FUNCTION_BLOCK ConveyorCTLServer (* Basic Function Block Type *)
  (* Standard: 61499-2 *)
  (* Version 0.2, 2003-12-04, JHC, Rockwell Automation, Renamed for better indexing. *)
  (* Version 0.1, 2002-11-05, JHC, Rockwell Automation, Corrected missing ST element in Algorithm REQ. *)
  (* Version 0.0, 2000-05-30, JHC, Rockwell Automation *)
  (* Compiler header: package fb.rt.cs725; *)
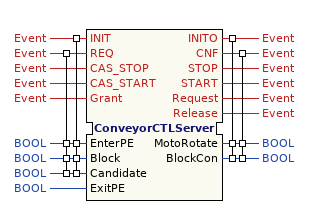
  EVENT_INPUT
    INIT WITH EnterPE, Block, Candidate; (* Initialization Request *)
    REQ WITH EnterPE, Block, Candidate; (* Normal Execution Request *)
    CAS_STOP;
    CAS_START;
    Grant;
  END_EVENT
  EVENT_OUTPUT
    INITO WITH MotoRotate, BlockCon; (* Initialization Confirm *)
    CNF WITH MotoRotate, BlockCon; (* Execution Confirmation *)
    STOP;
    START;
    Request;
    Release;
  END_EVENT
  VAR_INPUT
    EnterPE : BOOL; (* Input event qualifier *)
    Block : BOOL;
    Candidate : BOOL;
    ExitPE : BOOL;
  END_VAR
  VAR_OUTPUT
    MotoRotate : BOOL; (* Output event qualifier *)
    BlockCon : BOOL;
  END_VAR
  VAR
    lastPE : BOOL := 1;
    lastBlock : BOOL := 0;
  END_VAR
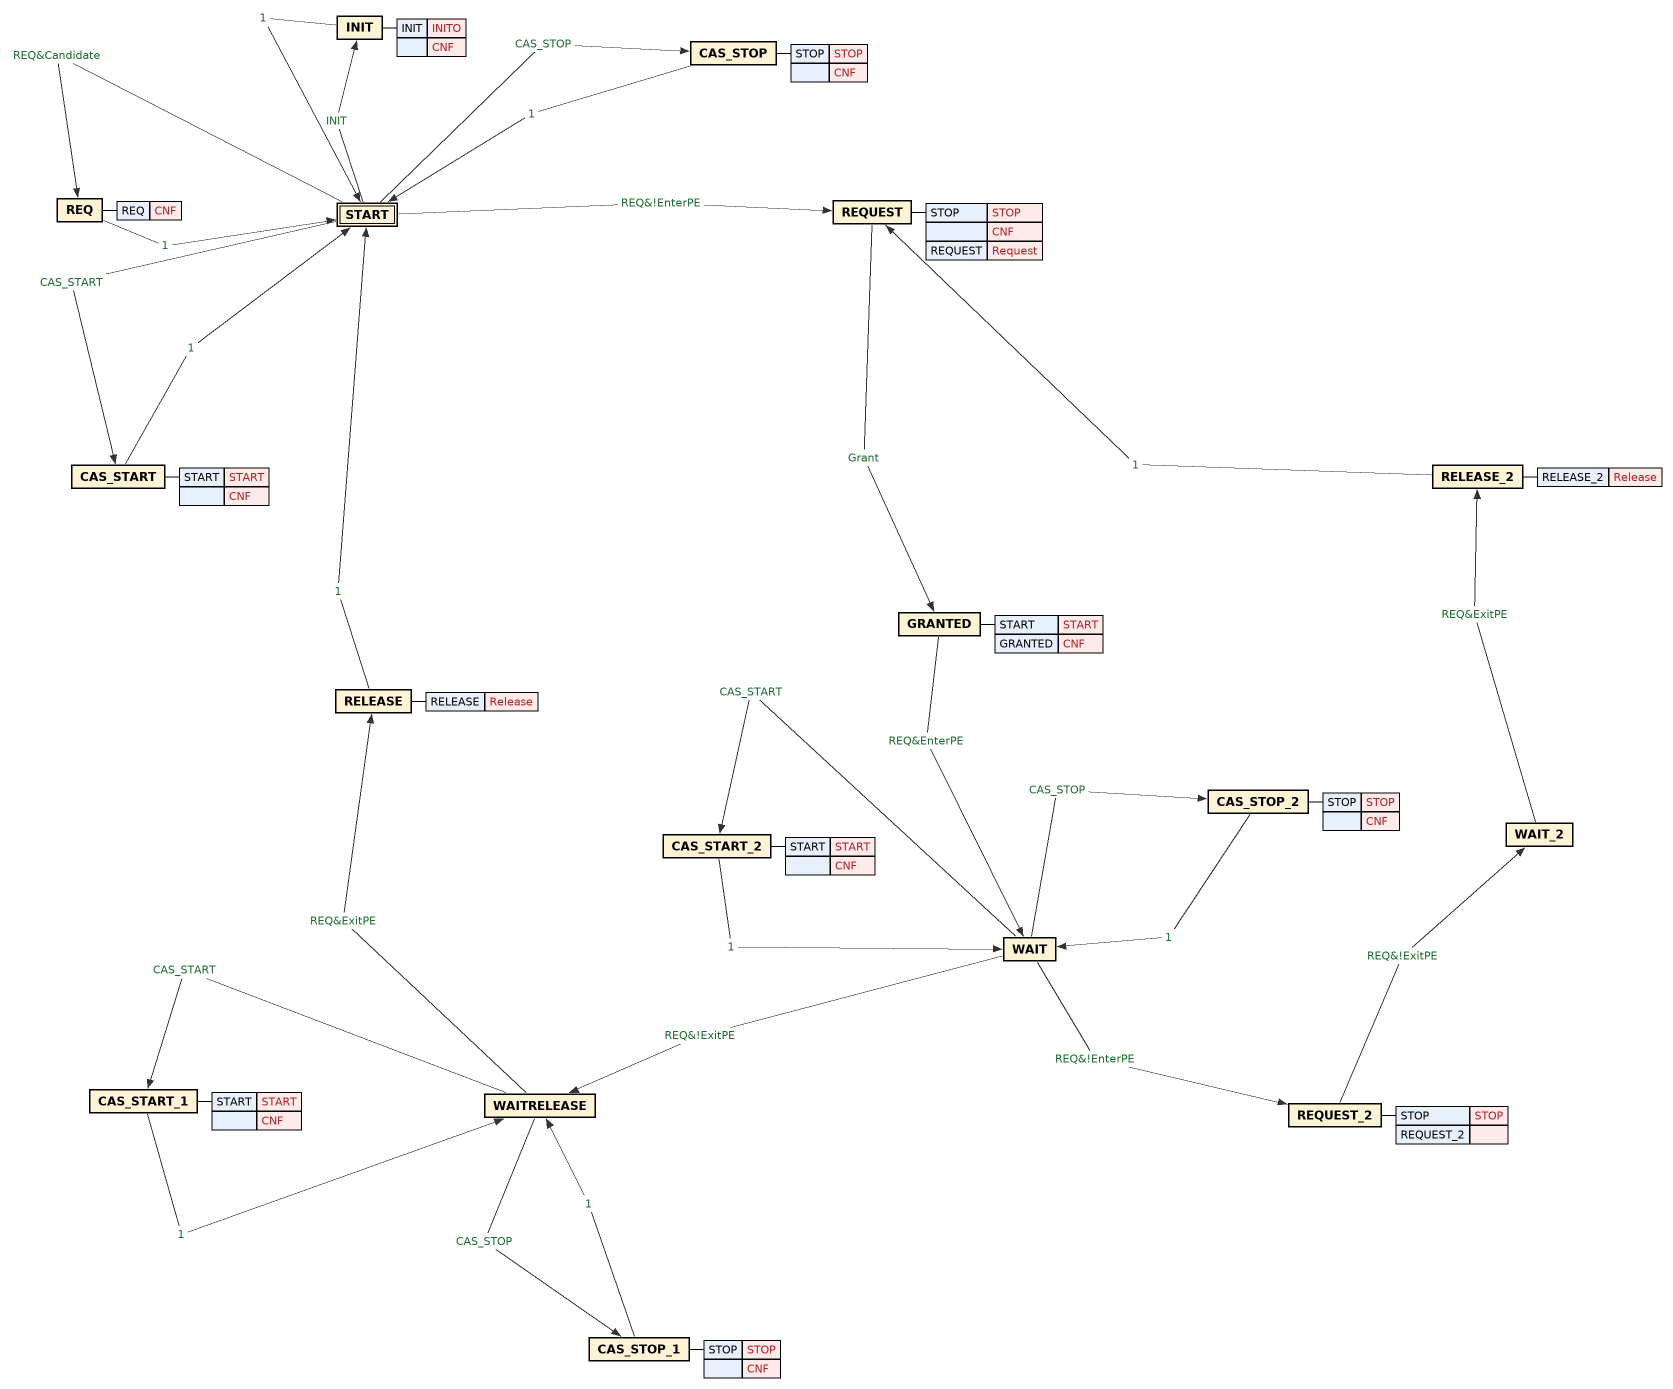
  EC_STATES
    START; (* Initial State *)
    INIT : INIT -> INITO, -> CNF; (* Initialization *)
    REQ : REQ -> CNF; (* Normal execution *)
    CAS_START : START -> START, -> CNF;
    CAS_STOP : STOP -> STOP, -> CNF;
    REQUEST : STOP -> STOP, -> CNF, REQUEST -> Request;
    GRANTED : START -> START, GRANTED -> CNF;
    RELEASE : RELEASE -> Release;
    WAIT;
    REQUEST_2 : STOP -> STOP, REQUEST_2;
    RELEASE_2 : RELEASE_2 -> Release;
    WAITRELEASE;
    WAIT_2;
    CAS_STOP_1 : STOP -> STOP, -> CNF;
    CAS_STOP_2 : STOP -> STOP, -> CNF;
    CAS_START_2 : START -> START, -> CNF;
    CAS_START_1 : START -> START, -> CNF;
  END_STATES
  EC_TRANSITIONS
    START TO INIT := INIT;
    INIT TO START := 1;
    START TO REQ := REQ&Candidate;
    REQ TO START := 1;
    START TO CAS_START := CAS_START;
    CAS_START TO START := 1;
    START TO CAS_STOP := CAS_STOP;
    CAS_STOP TO START := 1;
    REQUEST TO GRANTED := Grant;
    WAIT TO WAITRELEASE := REQ&!ExitPE;
    RELEASE TO START := 1;
    START TO REQUEST := REQ&!EnterPE;
    GRANTED TO WAIT := REQ&EnterPE;
    WAIT TO REQUEST_2 := REQ&!EnterPE;
    REQUEST_2 TO WAIT_2 := REQ&!ExitPE;
    RELEASE_2 TO REQUEST := 1;
    WAITRELEASE TO RELEASE := REQ&ExitPE;
    WAIT_2 TO RELEASE_2 := REQ&ExitPE;
    WAITRELEASE TO CAS_STOP_1 := CAS_STOP;
    CAS_STOP_1 TO WAITRELEASE := 1;
    WAIT TO CAS_STOP_2 := CAS_STOP;
    CAS_STOP_2 TO WAIT := 1;
    WAIT TO CAS_START_2 := CAS_START;
    CAS_START_2 TO WAIT := 1;
    WAITRELEASE TO CAS_START_1 := CAS_START;
    CAS_START_1 TO WAITRELEASE := 1;
  END_TRANSITIONS
  ALGORITHM INIT IN ST: (* Initialization algorithm *)
MotoRotate := TRUE;
Block := FALSE;
  END_ALGORITHM
  ALGORITHM REQ IN ST: (* Normally executed algorithm *)
IF Candidate THEN
IF lastPE !:= EnterPE THEN
IF NOT EnterPE THEN
BlockCon:= TRUE;
System.out.println("BlockCon = true");
ELSE
BlockCon:=FALSE;
System.out.println("BlockCon = false");
END_IF
lastPE := EnterPE;
END_IF
IF lastBlock !:= Block THEN
IF Block THEN
STOP.serviceEvent(this);
MotoRotate := FALSE;
System.out.println("Cas Stop");
ELSE
START.serviceEvent(this);
MotoRotate := TRUE;
System.out.println("Cas Start");
END_IF
lastBlock := Block;
END_IF
END_IF
  END_ALGORITHM
  ALGORITHM START IN ST:
MotoRotate:=TRUE;
  END_ALGORITHM
  ALGORITHM STOP IN Java:
MotoRotate.value=false;
  END_ALGORITHM
  ALGORITHM REQUEST IN Java:
System.out.println("Request to Central Server");
  END_ALGORITHM
  ALGORITHM GRANTED IN Java:
System.out.println("Request granted for Critical Section 1");
  END_ALGORITHM
  ALGORITHM REQUEST_2 IN Java:
System.out.println("Request 2nd");
  END_ALGORITHM
  ALGORITHM RELEASE_2 IN Java:
System.out.println("2nd Release token to Central Server");
  END_ALGORITHM
  ALGORITHM RELEASE IN Java:
System.out.println("Release token to Central Server");
  END_ALGORITHM
END_FUNCTION_BLOCK
